FUNCTION F_RaiseAlarmAndSetFlags : BOOL
VAR_IN_OUT
    fbAlarm    : FB_TcAlarm; //Alarm to be raised
    bErrorFlag : BOOL;       //Error flag to set (VAR_IN_OUT, put the variable you want the function to SET here)
    nErrorID   : UDINT;      //Error ID to set (VAR_IN_OUT, put the variable you want the function to SET here) - Will be set using the ID of the given fbAlarm
END_VAR

bErrorFlag := TRUE;
nErrorID   := fbAlarm.nEventId;

fbAlarm.Raise(0);

END_FUNCTION

(* stored: Version 1.1.0.1, ProductVersion 3.1.4024.11
   POU F_RaiseAlarmAndSetFlags: Id {18d943ce-984b-4d83-a2cd-d13434a0acee}, SpecialFunc None *)
